{attribute 'OPC.UA.DA.StructuredType' := '1'}
TYPE ST_BufferStorageState :
STRUCT
	fUpperTemperature : REAL;
	fMidTemperature : REAL;
	fLowerTemperature : REAL;
END_STRUCT
END_TYPE

(* stored: Version 1.1.0.1, ProductVersion 3.1.4024.10
   DUT ST_BufferStorageState: Id {f1cfeddc-16fe-4dea-9294-ce50413afc83} *)
